// TwinCAT 3 PLC project Lamppu8
// ProgramVersion: 3.1.4026.10
// CompilerDefines: VISU_USEPROPERTYINFO
// libraries:
//   Tc2_Standard, * (Beckhoff Automation GmbH)
//   Tc2_System, * (Beckhoff Automation GmbH)
// project tree:
//   / GlobalTextList.TcGTLO, PlcTask.TcTTO, Visualization Manager.TcVMO (not stored)
//   POUs/ MAIN.TcPOU
//   VISUs/ Visualization.TcVIS
// real-time tasks:
//   TASK PlcTask: cycle T#10ms, priority 20, ADS port 350

CONFIGURATION Lamppu8
    RESOURCE PLC ON TwinCAT3
        TASK PlcTask(INTERVAL := T#10ms, PRIORITY := 20);
        PROGRAM MAIN WITH PlcTask : MAIN;
    END_RESOURCE
END_CONFIGURATION

// ---- POUs/MAIN.TcPOU
PROGRAM MAIN
VAR
	_Button1	:BOOL;
	_Button2	:BOOL;
	_LampR		:BOOL; //Red light
	_LampY		:BOOL; //Yellow light
	_LampG		:BOOL; //Green light
END_VAR


//This lamp program turns three lights on and off. If button 1 is pushed,
//the red light comes on, if button 2 is pushed, the yellow light comes on,
//if both buttons are pushed, the green light comes on, and if neither button
//is pushed, no lights are on. This is the 8th exercise of the book, exercises
//3-7 were skipped since they are more or less the same as this one and the
//first two.

IF _Button1 AND NOT _Button2 THEN
	_LampR := TRUE;
	
	_LampG := FALSE;
	_LampY := FALSE;
ELSIF _Button2 AND NOT _Button1 THEN
	_LampY := TRUE;
	
	_LampG := FALSE;
	_LampR := FALSE;
ELSIF _Button1 AND _Button2 THEN
	_LampG := TRUE;
	
	_LampY := FALSE;
	_LampR := FALSE;
ELSE
	_LampG := FALSE;
	_LampY := FALSE;
	_LampR := FALSE;
END_IF

END_PROGRAM

// ---- GlobalTextList.TcGTLO
TEXTLIST GlobalTextList
  443 = 'Button 1'
  332 = 'Button 2'
END_TEXTLIST

// ---- VISUs/Visualization.TcVIS
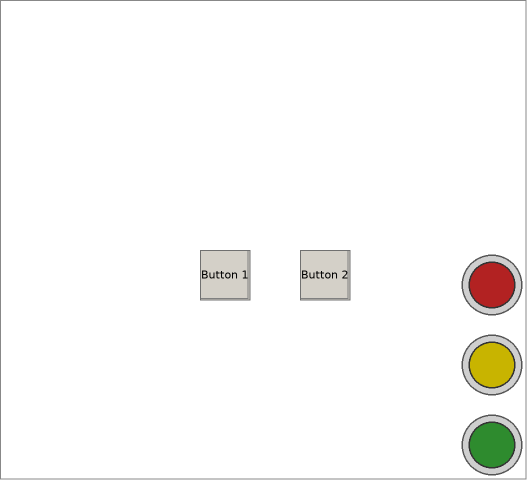
VISUALIZATION Visualization  // 527x480
    Button (200,250 50x50), "Button 1"
        OnMouseClick: toggle MAIN._Button1
    Button (300,250 50x50), "Button 2"
        OnMouseClick: toggle MAIN._Button2
    Lamp1 (457,250 70x70), variable: MAIN._LampR, style: Lamp-Lamp1-Red
    Lamp1 (457,330 70x70), variable: MAIN._LampY, style: Lamp-Lamp1-Yellow
    Lamp1 (457,410 70x70), variable: MAIN._LampG, style: Lamp-Lamp1-Green
END_VISUALIZATION
